FUNCTION_BLOCK FB_PressureGroup IMPLEMENTS I_PressureGroup
VAR_INPUT
    fPressureLimitLow: REAL := 1.0; //Minimum pressure limit
    fPressureLimitHigh: REAL := 6.0; //Maximum pressure limit
    tPressureOutOfRange: TIME := T#15S; //Time limit pressure is out of range
    fRawHigh: REAL := 30518.0; //Highest value for the Raw value
    fRawLow: REAL := 0.0; //Lowest value for the Raw value
    fScaledHigh: REAL := 10.0; //Highest value for the Scaled value 10 bar
    fScaledLow: REAL := 0.0; //Lowest value for the Scaled value 0 bar
END_VAR
VAR_IN_OUT CONSTANT
    nAirPressureSensorRaw: INT; //Raw value from analog air pressure sensor
END_VAR
VAR
    _fScaledPressureValue: REAL;
    tonTimerPressureLow: TON := (Q := TRUE);
    tonTimerPressureHigh: TON := (Q := TRUE);
END_VAR

_fScaledPressureValue := mScalePressureValue(nRawValue := nAirPressureSensorRaw);

tonTimerPressureLow(
    IN := _fScaledPressureValue < fPressureLimitLow,
    PT := tPressureOutOfRange);

tonTimerPressureHigh(
    IN := _fScaledPressureValue > fPressureLimitHigh,
    PT := tPressureOutOfRange);

PROPERTY bPressureHigh : BOOL
GET
bPressureHigh := tonTimerPressureHigh.Q;
END_GET
END_PROPERTY

PROPERTY bPressureLow : BOOL
GET
bPressureLow := tonTimerPressureLow.Q;
END_GET
END_PROPERTY

PROPERTY fScaledPressureValue : REAL
GET
fScaledPressureValue := _fScaledPressureValue;
END_GET
END_PROPERTY

METHOD PUBLIC mScalePressureValue : REAL
VAR_INPUT
    nRawValue: INT; //Raw value from the Terminal
END_VAR
VAR
    rGradient: REAL; //Internal variable to calculate gradient of the slope
    rOffset: REAL; //Internal variable to calculate the offset value
END_VAR
rGradient:= (fScaledHigh - fScaledLow)/(fRawHigh - fRawLow);
rOffset:= fScaledHigh - rGradient * fRawHigh;
mScalePressureValue:= rGradient * nRawValue + rOffset;
END_METHOD

END_FUNCTION_BLOCK

(* stored: Version 1.1.0.1
   POU FB_PressureGroup: Id {bdc1d7c0-6b5c-06bf-358c-d7d1869947c6}, SpecialFunc None
   Property bPressureHigh: Id {a98d5871-a004-082f-2621-3184809d1573}
   Get Get: Id {f3b4e553-8860-0192-16e6-469b74f61a51}
   Property bPressureLow: Id {be51e195-fa7f-0ccc-3811-074a1e15914f}
   Get Get: Id {cb05adcf-d57e-0d22-1095-76ebd24bf9b5}
   Property fScaledPressureValue: Id {ea8dfccc-e203-05f0-3d29-bbe5890bd9eb}
   Get Get: Id {3ebff06d-3e02-0ee2-1268-04c0624560bf}
   Method mScalePressureValue: Id {b7519c62-7156-0d37-0443-eeecc8fc8823} *)
